// TIA Portal V18 export
DATA_BLOCK "Servo Control"   // DB336
{ S7_Optimized_Access := 'TRUE' }
VERSION : 0.1
// stored: AutoNumber false, DBAccessibleFromOPCUA true, IsOnlyStoredInLoadMemory false, IsRetainMemResEnabled false, IsWriteProtectedInAS false, MemoryReserve 100
   VAR
      "A" : Struct
         "Power On" : Bool;
         Reset : Bool;
         Restart : Bool;
         "Speed input" : Real;
         Velocity : Real;
         "Power Error" : Bool;
         "drive error" : Bool;
         "Communication Error" : Bool;
         "Actual Velocity" : Real;
         RPM : Real;
      END_STRUCT;
      "B" : Struct
         "Power On" : Bool;
         Reset : Bool;
         Restart : Bool;
         "Speed input" : Real;
         Velocity : Real;
         "Power Error" : Bool;
         "drive error" : Bool;
         "Communication Error" : Bool;
         "Actual Velocity" : Real;
         RPM : Real;
      END_STRUCT;
      Mixer : Struct
         "Power On" : Bool;
         Reset : Bool;
         Restart : Bool;
         "Speed input" : Real;
         Velocity : Real;
         "Power Error" : Bool;
         "drive error" : Bool;
         "Communication Error" : Bool;
         "Actual Velocity" : Real;
         RPM : Real;
      END_STRUCT;
   END_VAR
BEGIN
END_DATA_BLOCK
